FUNCTION_BLOCK E_CTD (* Event-Driven Down Counter *)
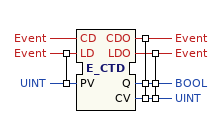
  EVENT_INPUT
    CD; (* Count Down *)
    LD WITH PV; (* Load counter value *)
  END_EVENT
  EVENT_OUTPUT
    CDO WITH Q, CV; (* Count Down Output Event *)
    LDO WITH Q, CV; (* Reset Output Event *)
  END_EVENT
  VAR_INPUT
    PV : UINT; (* Preset Value *)
  END_VAR
  VAR_OUTPUT
    Q : BOOL; (* CV <= 0 *)
    CV : UINT; (* Counter Value *)
  END_VAR
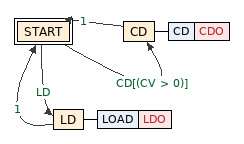
  EC_STATES
    START;
    CD : CD -> CDO;
    LD : LOAD -> LDO;
  END_STATES
  EC_TRANSITIONS
    START TO CD := CD[(CV > 0)];
    CD TO START := 1;
    START TO LD := LD;
    LD TO START := 1;
  END_TRANSITIONS
  ALGORITHM CD IN ST:
CV := CV - 1;
Q := (CV = 0);
  END_ALGORITHM
  ALGORITHM LOAD IN ST:
CV := PV;
Q:= (CV = 0);
  END_ALGORITHM
END_FUNCTION_BLOCK
